{attribute addProperty BoxType "EPP3752-0000-0017"}
{attribute addProperty Id "AI_Inputs_ChannelAT %I*ARRAY[0..5] OF AI_Inputs_Channel_83E63207192240WcStateAT %I*WcState_F855686C1620InfoDataAT %I*InfoData_BC63D37F80100"}
{attribute addProperty CRC "2876859799"}
{attribute addProperty SizeInBites "288"}
{attribute addProperty SizeInBytes "36"}
TYPE EPP3752_AEF24F9C :
STRUCT
	{attribute addProperty Name "AI_Inputs_Channel"}
	AI_Inputs_Channel : ARRAY[0..5] OF AI_Inputs_Channel_83E63207;
	{attribute addProperty Name "WcState"}
	WcState : WcState_F855686C;
	{attribute addProperty Name "InfoData"}
	InfoData : InfoData_BC63D37F;
END_STRUCT
END_TYPE

(* stored: Version 1.2.0.0, ProductVersion 3.1.4024.9
   DUT EPP3752_AEF24F9C: Id {d7f104c1-21b3-44bb-b1f6-91e83ee2149c} *)
